// Copyright (c) 2024 Loupe (https://loupe.team), provided under the MIT License.

INTERFACE IPLCopenCallRemote EXTENDS __SYSTEM.IQueryInterface


METHOD ReportAborted : BOOL
VAR_INPUT
END_VAR
END_METHOD


METHOD ReportErrored : BOOL
VAR_INPUT
  ID : INT;
END_VAR
END_METHOD


METHOD ReportFinished : BOOL
VAR_INPUT
END_VAR
END_METHOD

END_INTERFACE

(* stored: Version 1.1.0.1
   Itf IPLCopenCallRemote: Id {6aa201bf-eb14-40e6-82eb-dedd5645dc58}
   Method ReportAborted: Id {86840f40-10b0-4de0-ab69-6c5eb8f761fb}
   Method ReportErrored: Id {6b8dd4a3-2d32-4590-a313-c41aaa663229}
   Method ReportFinished: Id {bd57ce11-7e84-4c4a-bfa9-527eee6bb14e} *)
